FUNCTION_BLOCK CommFromMatlab2 (* Extracted Composite Function Block Type *)
  (* Version 5/20/2016, gulzha *)
  PACKAGE Main;
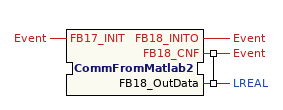
  EVENT_INPUT
    FB17_INIT; (* Initialization request event *)
  END_EVENT
  EVENT_OUTPUT
    FB18_INITO; (* Initialization Confirm *)
    FB18_CNF WITH FB18_OutData; (* Execution Confirmation *)
  END_EVENT
  VAR_OUTPUT
    FB18_OutData : LREAL;
  END_VAR
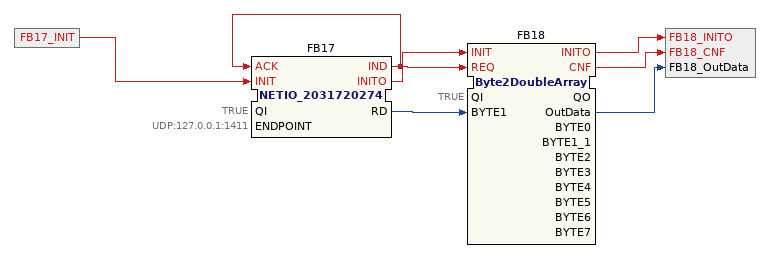
  FBS
    FB17 : NETIO_2031720274(QI := TRUE, ENDPOINT := UDP:127.0.0.1:1411); {SET_ATTRIBUTE(Configuration.GenericFBType.InterfaceParams, Runtime.IoCommon#I:=1;SD:BYTE[8];RD:BYTE[8])}
    FB18 : Byte2DoubleArray(QI := TRUE);
  END_FBS
  EVENT_CONNECTIONS
    FB17.IND TO FB17.ACK;
    FB17.INITO TO FB18.INIT;
    FB17.IND TO FB18.REQ;
    FB17_INIT TO FB17.INIT;
    FB18.INITO TO FB18_INITO;
    FB18.CNF TO FB18_CNF;
  END_CONNECTIONS
  DATA_CONNECTIONS
    FB17.RD TO FB18.BYTE1;
    FB18.OutData TO FB18_OutData;
  END_CONNECTIONS
END_FUNCTION_BLOCK
